// SIMATIC STEP 7 (V5.x) project dry_cooler
// CPU: CPU313(1)
// station: P_ADR_BUS
// station: Hardware
// station: SIMATIC 300 Station
// station: P_ADR_BUS
// station: Configuration
// program: S7 Program(1)

SYMBOL_TABLE
"DBData"	DB 1	DB 1
"DB_Alarm"	DB 2	DB 2	// Db alarmes
"Run Time Animation"	DB 3	DB 3	// Animaçoes
"DBAnalog"	DB 64	DB 64
"DB_Temperature"	DB 100	DB 100	// DB Tratamento analogico
"DB HMI Funtions"	DB 101	DB 101
"Sensores"	FB 105	FB 105
"Analog_Trated"	FC 1	FC 1	// Analog_trated
"Input_Trated"	FC 2	FC 2	// Tratatemto das entradas
"Output_Trated"	FC 3	FC 3	// Tratamento das saidas
"Inputs"	FC 4	FC 4	// Inputs
"Outputs"	FC 5	FC 5	// Outputs
"Pump_Logic"	FC 6	FC 6
"Acionaqamento Ventilador"	FC 7	FC 7
"New Analog"	FC 10	FC 10
"Tratamento_Inputs"	FC 100	FC 100
"Tratamento Saida"	FC 101	FC 101
"SCALE_1"	FC 105	FC 105	// Scaling 1
"Transmissores_Analogicos"	FC 106	FC 106
"SCALE_2"	FC 205	FC 205	// Scaling 2
"Animation_HMI"	FC 255	FC 255
"SCALE_3"	FC 305	FC 305	// Scaling 2
"SCALE_4"	FC 405	FC 405	// Scaling 4
"SCALE_5"	FC 505	FC 505	// Scaling 5
"SCALE_6"	FC 605	FC 605	// Scaling 6
"SCALE_7"	FC 705	FC 705	// Scaling 7
"SCALE_8"	FC 805	FC 805	// Scaling 8
"Pump1_On"	I 4.0	BOOL	// Button On Pump1
"Pump1_Off"	I 4.1	BOOL	// Button Off Pump1
"Pump_2_On"	I 4.2	BOOL	// Button On Pump2
"Puymp2_Off"	I 4.3	BOOL	// Button Off Pump2
"Fan1_On"	I 4.4	BOOL	// Button On Fan1
"Fan1_Off"	I 4.5	BOOL	// Button Off Fan1
"Fan2_On"	I 4.6	BOOL	// Button On Fan2
"Fan2_Off"	I 4.7	BOOL	// Button Off Fan2
"AdiabaticPump_On"	I 5.0	BOOL	// Button On Adb
"AdiabaticPump_Off"	I 5.1	BOOL	// Button Off Adb
"Emergency"	I 5.2	BOOL	// Emergency Button
"Manual"	I 5.3	BOOL	// Manual Switch
"Auto"	I 5.4	BOOL	// Auto Switch
"InSpare1"	I 5.5	BOOL	// Spare 1
"InSpare2"	I 5.6	BOOL	// Spare2
"InSpare3"	I 5.7	BOOL	// Spare3
"CircuitBreakerPump1"	I 8.0	BOOL	// Feedback CB Pump1
"CircuitBrakerPump2"	I 8.1	BOOL	// Feedback CB Pump2
"CircuitBreaker Fan1"	I 8.2	BOOL	// Feedback CB Fan1
"CircuitBraekerFan2"	I 8.3	BOOL	// Feedback CB Fan2
"CircuitBreakerAdbPump"	I 8.4	BOOL	// Feedback CB Adiabatic Pump
"ContactorPump1"	I 8.5	BOOL	// Feedback state contactor pump 1
"ContactorPump2"	I 8.6	BOOL	// Feedback state contactor pump 2
"Contacort.Fan1"	I 8.7	BOOL	// Feedback state contactor fan 1
"ContactorFan2"	I 9.0	BOOL	// Feedback state contactor fan2
"ContactorAdb"	I 9.1	BOOL	// Feedback state contactor adb pump
"FlowSwitch"	I 9.2	BOOL	// Flow Switch signal
"LevelSwitch"	I 9.3	BOOL	// Level switch
"InSpare4"	I 9.4	BOOL	// Spare 4
"InSpare5"	I 9.5	BOOL	// Spare 5
"InSpare6"	I 9.6	BOOL	// Spare 6
"InSpare7"	I 9.7	BOOL	// Spare 7
"Aux_Pump1On"	M 4.0	BOOL	// Aux input pump 1 on
"Aux_Pump1Off"	M 4.1	BOOL	// Aux input pump 1 off
"Aux_Pump2On"	M 4.2	BOOL	// Aux input pump 2 on
"Aux_Pump2Off"	M 4.3	BOOL	// Aux input pump 2 off
"Aux_Fan1On"	M 4.4	BOOL	// Aux input fan 1 on
"Aux_Fan1Off"	M 4.5	BOOL	// Aux input fan 1 off
"Aux_Fan2On"	M 4.6	BOOL	// Aux input fan 2on
"Aux_Fan2Off"	M 4.7	BOOL	// Aux input fan 2 off
"Aux_AdbOn"	M 5.0	BOOL	// Aux input adiabatic on
"Aux_AdbOff"	M 5.1	BOOL	// Aux input adiabatic off
"Aux_Emergency"	M 5.2	BOOL	// Aux input emergency button
"Aux_Manual"	M 5.3	BOOL	// Aux input manual Switch
"Aux_Automatic"	M 5.4	BOOL	// Aux input automatic switch
"Aux_InSpare1"	M 5.5	BOOL	// Aux input spare1
"Aux_InSpare2"	M 5.6	BOOL	// Aux input spare2
"Aux_InSpare3"	M 5.7	BOOL	// Aux input spare3
"Aux_CBPump1"	M 8.0	BOOL	// Aux input circuit breaker pump 1
"Aux_CBPump2"	M 8.1	BOOL	// Aux input circuit breaker pump2
"Aux_CBFan1"	M 8.2	BOOL	// Aux input circuit breaker fan 1
"Aux_CBFan2"	M 8.3	BOOL	// Aux input circuit breaker fan 2
"Aux_CBAdbPump"	M 8.4	BOOL	// Aux input circuit breaker adiabatic
"Aux_FeedPump1"	M 8.5	BOOL	// Aux input feedback contactor pump 1
"Aux_FeedPump2"	M 8.6	BOOL	// Aux input feedback contactor pump 2
"Aux_FeedFan1"	M 8.7	BOOL	// Aux input feedback contactor fan 1
"Aux_FeedFan2"	M 9.0	BOOL	// Aux input feedback contactor fan 2
"Aux_FeedAdbPump"	M 9.1	BOOL	// Aux input feedbcak contactor adiabatic
"Aux_FlowSwitch"	M 9.2	BOOL	// Aux input flow switch
"Aux_LevelSwitch"	M 9.3	BOOL	// Aux input level switch
"Aux_InSpare4"	M 9.4	BOOL	// Aux input spare 4
"Aux_InSpare5"	M 9.5	BOOL	// Aux input spare 5
"Aux_InSpare6"	M 9.6	BOOL	// Aux input spare 6
"Aux_InSpare7"	M 9.7	BOOL	// Auxiliar Input spare 7
"OnAutomaticPump1"	M 10.0	BOOL	// Start pump 1 Automatic
"OnManualPump1"	M 10.1	BOOL	// Start Pump 1 Manual
"Flow Fault"	M 10.2	BOOL	// Water flow in fault pump 1
"Aux_RelayWaterPump1"	M 12.0	BOOL	// Aux out relay pump 1
"Aux_RelayWaterPump2"	M 12.1	BOOL	// Aux out relay pump2
"Aux_RelayFan1"	M 12.2	BOOL	// Aux out relay fan 1
"Aux_RelayFan2"	M 12.3	BOOL	// Aux out relay fan 2
"Aux_RelayAdbPump"	M 12.4	BOOL	// Aux out relay adiabatic pump
"Aux_OutSpare1"	M 12.5	BOOL	// Aux out spare 1
"Aux_OutSpare2"	M 12.6	BOOL	// Aux out spare 2
"Aux_OutSpare3"	M 12.7	BOOL	// Aux out spare 3
"Aux_OutSpare4"	M 13.0	BOOL	// Aux out spare 4
"Aux_OutSpare5"	M 13.1	BOOL	// Aux out spare 5
"Aux_OutSpare6"	M 13.2	BOOL	// Aux out spare 6
"Aux_OutSpare7"	M 13.3	BOOL	// Aux out spare 7
"Aux_HornBuzzer"	M 13.4	BOOL	// Aux out horn buzzer
"Aux_AdiabaticSolenoid"	M 13.5	BOOL	// Aux out adiabatic solenoid
"Aux_LampPump1On"	M 13.6	BOOL	// Aux out lamp pump 1 on
"Aux_LampPump1Fault"	M 13.7	BOOL	// Aux out lamp pump 1 fault
"Aux_LampPump2On"	M 16.0	BOOL	// Aux out lamp pump 2 on
"Aux_LampPump2Fault"	M 16.1	BOOL	// Aux out lamp pump 2 fault
"Aux_LampFan1On"	M 16.2	BOOL	// Aux out lamp fan 1 on
"Aux_LampFan1Fault"	M 16.3	BOOL	// Aux out lamp fan 1 fault
"Aux_LampFan2On"	M 16.4	BOOL	// Aux out lamp fan 2 on
"Aux_LampFan2Fault"	M 16.5	BOOL	// Aux out lamp fan 2 fault
"Aux_LampAdiabaticOn"	M 16.6	BOOL	// Aux out lamp adiabatic on
"Aux_LampAdiabaticFault"	M 16.7	BOOL	// Aux out lamp adiabatic fault
"DI_Input"	MW 2	WORD
"R_Input"	MW 4	WORD
"Cycle Execution"	OB 1	OB 1
"Loss of Rack Fault"	OB 86	OB 86
"Complete Restart"	OB 100	OB 100
"Temp_Input"	PIW 256	WORD	// Temp_Input
"Temp_Output"	PIW 258	WORD	// Temp_Output
"RelayWaterPump1"	Q 12.0	BOOL	// Relay water pum 1
"RelayWaterPump2"	Q 12.1	BOOL	// Relay water Pump 2
"RelayFan1"	Q 12.2	BOOL	// Relay fan 1
"RelayFan2"	Q 12.3	BOOL	// Relay fan 2
"RelayAdiabaticPump"	Q 12.4	BOOL	// Relay adiabatic pump
"OutSpare1"	Q 12.5	BOOL	// Out Spare1
"OutSpare2"	Q 12.6	BOOL	// Out Spare 2
"OutSpare3"	Q 12.7	BOOL	// Out Spare 3
"OutSpare4"	Q 13.0	BOOL	// Out Spare 4
"OutSpare5"	Q 13.1	BOOL	// Out Spare 5
"OutSpare6"	Q 13.2	BOOL	// Out Spare 6
"OutSpare7"	Q 13.3	BOOL	// Out Spare 7
"HornBuzzer"	Q 13.4	BOOL	// Horn Buzzer
"RelayAdbSolenoid"	Q 13.5	BOOL	// Relay adiabatic solenoid
"LightOnPump1"	Q 13.6	BOOL	// Light on pump 1
"LightFaultPump1"	Q 13.7	BOOL	// Light fault pump 1
"LightOnPump2"	Q 16.0	BOOL	// Light on pump 2
"LightFaultPump2"	Q 16.1	BOOL	// Light fault pump 2
"LightOnFan1"	Q 16.2	BOOL	// Light on fan 1
"LightFaultFan1"	Q 16.3	BOOL	// Light fault fan 1
"LightOnFan2"	Q 16.4	BOOL	// Light on fan 2
"LightFaultFan2"	Q 16.5	BOOL	// Light fault fan 2
"LightOnAdb"	Q 16.6	BOOL	// Light on adiabatic
"LightFaultAdb"	Q 16.7	BOOL	// Light fault adiabatic
"Timer Water Flow"	T 0	TIMER
"Factor And ValueSensor"	VAT 1	
END_SYMBOL_TABLE

FUNCTION "Analog_Trated" : VOID	// FC 1
VERSION : 0.1
BEGIN
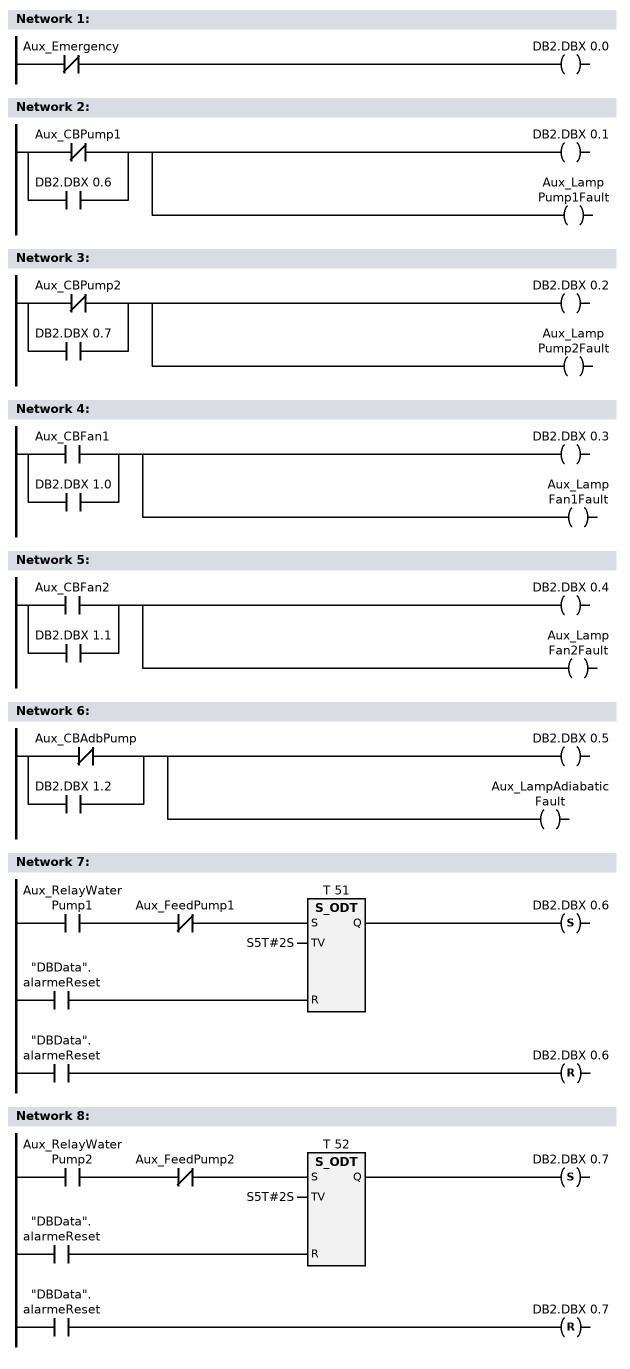
NETWORK
TITLE =
      AN    "Aux_Emergency";
      =     DB2.DBX 0.0;
NETWORK
TITLE =
      ON    "Aux_CBPump1";
      O     DB2.DBX 0.6;
      =     DB2.DBX 0.1;
      =     "Aux_LampPump1Fault";
NETWORK
TITLE =
      ON    "Aux_CBPump2";
      O     DB2.DBX 0.7;
      =     DB2.DBX 0.2;
      =     "Aux_LampPump2Fault";
NETWORK
TITLE =
      O     "Aux_CBFan1";
      O     DB2.DBX 1.0;
      =     DB2.DBX 0.3;
      =     "Aux_LampFan1Fault";
NETWORK
TITLE =
      O     "Aux_CBFan2";
      O     DB2.DBX 1.1;
      =     DB2.DBX 0.4;
      =     "Aux_LampFan2Fault";
NETWORK
TITLE =
      ON    "Aux_CBAdbPump";
      O     DB2.DBX 1.2;
      =     DB2.DBX 0.5;
      =     "Aux_LampAdiabaticFault";
NETWORK
TITLE =
      A(;
      A     "Aux_RelayWaterPump1";
      AN    "Aux_FeedPump1";
      L     S5T#2S;
      SD    T 51;
      A     "DBData".alarmeReset;
      R     T 51;
      NOP   0;
      NOP   0;
      A     T 51;
      );
      S     DB2.DBX 0.6;
      A     "DBData".alarmeReset;
      R     DB2.DBX 0.6;
      NOP   0;
NETWORK
TITLE =
      A(;
      A     "Aux_RelayWaterPump2";
      AN    "Aux_FeedPump2";
      L     S5T#2S;
      SD    T 52;
      A     "DBData".alarmeReset;
      R     T 52;
      NOP   0;
      NOP   0;
      A     T 52;
      );
      S     DB2.DBX 0.7;
      A     "DBData".alarmeReset;
      R     DB2.DBX 0.7;
      NOP   0;
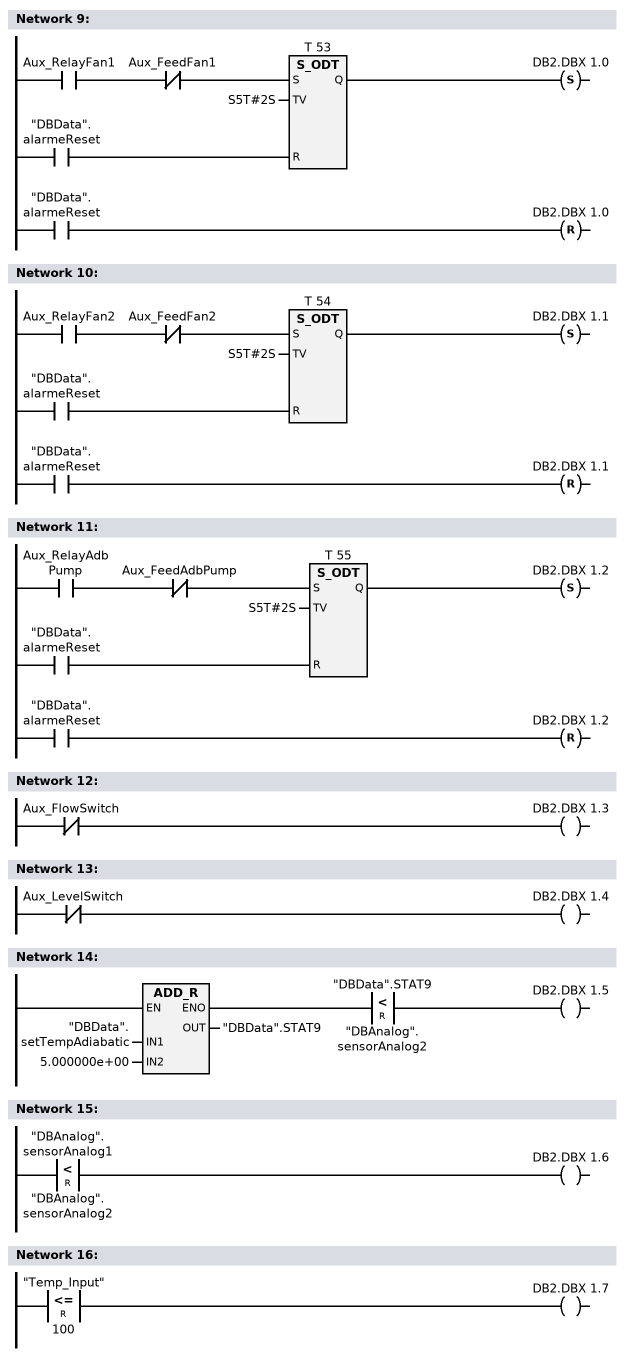
NETWORK
TITLE =
      A(;
      A     "Aux_RelayFan1";
      AN    "Aux_FeedFan1";
      L     S5T#2S;
      SD    T 53;
      A     "DBData".alarmeReset;
      R     T 53;
      NOP   0;
      NOP   0;
      A     T 53;
      );
      S     DB2.DBX 1.0;
      A     "DBData".alarmeReset;
      R     DB2.DBX 1.0;
      NOP   0;
NETWORK
TITLE =
      A(;
      A     "Aux_RelayFan2";
      AN    "Aux_FeedFan2";
      L     S5T#2S;
      SD    T 54;
      A     "DBData".alarmeReset;
      R     T 54;
      NOP   0;
      NOP   0;
      A     T 54;
      );
      S     DB2.DBX 1.1;
      A     "DBData".alarmeReset;
      R     DB2.DBX 1.1;
      NOP   0;
NETWORK
TITLE =
      A(;
      A     "Aux_RelayAdbPump";
      AN    "Aux_FeedAdbPump";
      L     S5T#2S;
      SD    T 55;
      A     "DBData".alarmeReset;
      R     T 55;
      NOP   0;
      NOP   0;
      A     T 55;
      );
      S     DB2.DBX 1.2;
      A     "DBData".alarmeReset;
      R     DB2.DBX 1.2;
      NOP   0;
NETWORK
TITLE =
      AN    "Aux_FlowSwitch";
      =     DB2.DBX 1.3;
NETWORK
TITLE =
      AN    "Aux_LevelSwitch";
      =     DB2.DBX 1.4;
NETWORK
TITLE =
      A(;
      L     "DBData".setTempAdiabatic;
      L     5.000000e+00;
      +R;
      T     "DBData".STAT9;
      AN    OV;
      SAVE;
      CLR;
      A     BR;
      );
      A(;
      L     "DBData".STAT9;
      L     "DBAnalog".sensorAnalog2;
      <R;
      );
      =     DB2.DBX 1.5;
NETWORK
TITLE =
      L     "DBAnalog".sensorAnalog1;
      L     "DBAnalog".sensorAnalog2;
      <R;
      =     DB2.DBX 1.6;
NETWORK
TITLE =
      L     "Temp_Input";
      L     100;
      <=R;
      =     DB2.DBX 1.7;
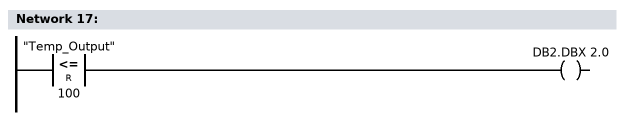
NETWORK
TITLE =
      L     "Temp_Output";
      L     100;
      <=R;
      =     DB2.DBX 2.0;
END_FUNCTION

FUNCTION "Input_Trated" : VOID	// FC 2
NAME : Inputs
VERSION : 0.1
BEGIN
// (block stored without names or comments; labels and parameter names are numbered)
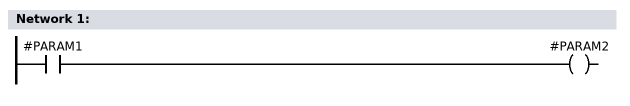
NETWORK
TITLE =
      A     #PARAM1;
      =     #PARAM2;
END_FUNCTION

FUNCTION "Output_Trated" : VOID	// FC 3
VERSION : 0.1
BEGIN
// (block stored without names or comments; labels and parameter names are numbered)
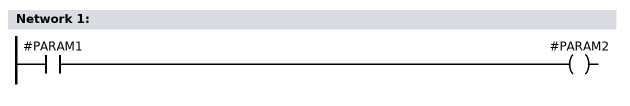
NETWORK
TITLE =
      A     #PARAM1;
      =     #PARAM2;
END_FUNCTION

FUNCTION "Inputs" : VOID	// FC 4
VERSION : 0.1
BEGIN
// (block stored without names or comments; labels and parameter names are numbered)
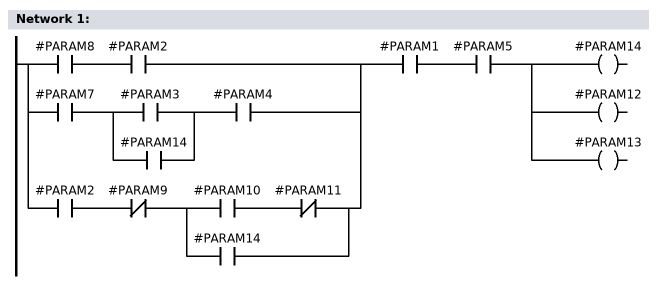
NETWORK
TITLE =
      A(;
      A     #PARAM8;
      A     #PARAM2;
      O;
      A     #PARAM7;
      A(;
      O     #PARAM3;
      O     #PARAM14;
      );
      A     #PARAM4;
      O;
      A     #PARAM2;
      AN    #PARAM9;
      A(;
      A     #PARAM10;
      AN    #PARAM11;
      O     #PARAM14;
      );
      );
      A     #PARAM1;
      A     #PARAM5;
      =     #PARAM14;
      =     #PARAM12;
      =     #PARAM13;
END_FUNCTION

FUNCTION "Outputs" : VOID	// FC 5
VERSION : 0.1
BEGIN
// (block stored without names or comments; labels and parameter names are numbered)
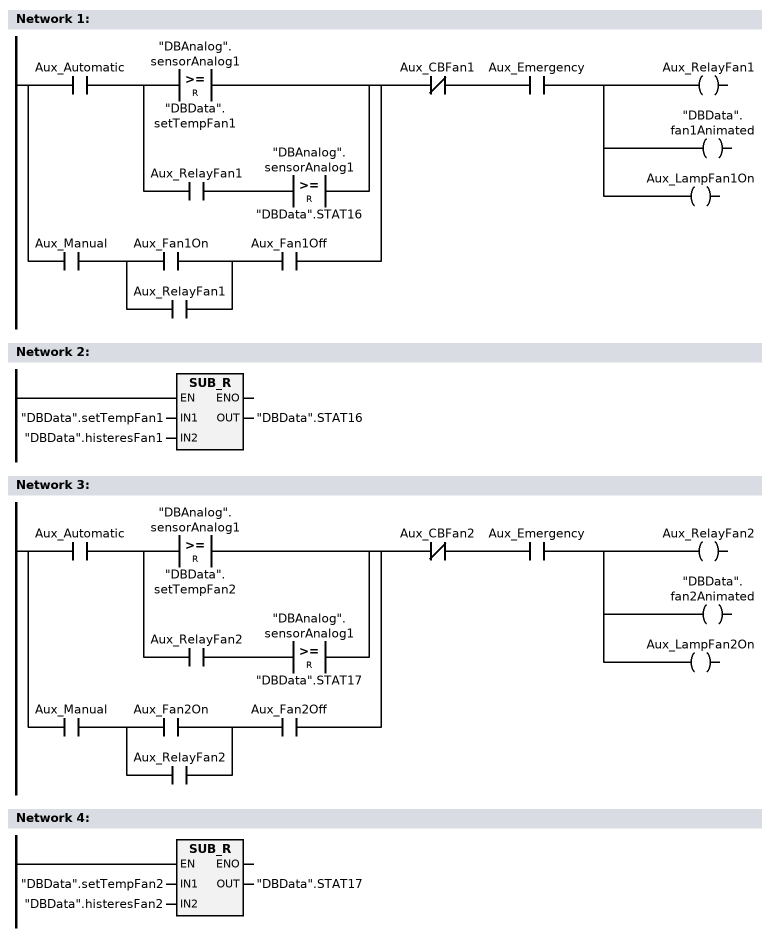
NETWORK
TITLE =
      A(;
      A     "Aux_Automatic";
      A(;
      O(;
      L     "DBAnalog".sensorAnalog1;
      L     "DBData".setTempFan1;
      >=R;
      );
      O;
      A     "Aux_RelayFan1";
      A(;
      L     "DBAnalog".sensorAnalog1;
      L     "DBData".STAT16;
      >=R;
      );
      );
      O;
      A     "Aux_Manual";
      A(;
      O     "Aux_Fan1On";
      O     "Aux_RelayFan1";
      );
      A     "Aux_Fan1Off";
      );
      AN    "Aux_CBFan1";
      A     "Aux_Emergency";
      =     "Aux_RelayFan1";
      =     "DBData".fan1Animated;
      =     "Aux_LampFan1On";
NETWORK
TITLE =
      L     "DBData".setTempFan1;
      L     "DBData".histeresFan1;
      -R;
      T     "DBData".STAT16;
      NOP   0;
NETWORK
TITLE =
      A(;
      A     "Aux_Automatic";
      A(;
      O(;
      L     "DBAnalog".sensorAnalog1;
      L     "DBData".setTempFan2;
      >=R;
      );
      O;
      A     "Aux_RelayFan2";
      A(;
      L     "DBAnalog".sensorAnalog1;
      L     "DBData".STAT17;
      >=R;
      );
      );
      O;
      A     "Aux_Manual";
      A(;
      O     "Aux_Fan2On";
      O     "Aux_RelayFan2";
      );
      A     "Aux_Fan2Off";
      );
      AN    "Aux_CBFan2";
      A     "Aux_Emergency";
      =     "Aux_RelayFan2";
      =     "DBData".fan2Animated;
      =     "Aux_LampFan2On";
NETWORK
TITLE =
      L     "DBData".setTempFan2;
      L     "DBData".histeresFan2;
      -R;
      T     "DBData".STAT17;
      NOP   0;
END_FUNCTION

FUNCTION "Pump_Logic" : VOID	// FC 6
VERSION : 0.1
BEGIN
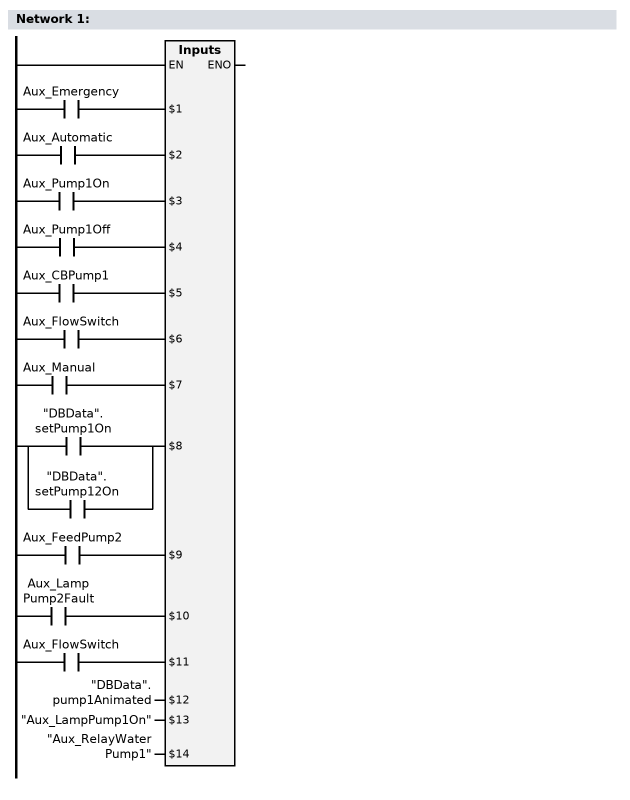
NETWORK
TITLE =
      A     "Aux_Emergency";
      =     L 0.0;
      BLD   103;
      A     "Aux_Automatic";
      =     L 0.1;
      BLD   103;
      A     "Aux_Pump1On";
      =     L 0.2;
      BLD   103;
      A     "Aux_Pump1Off";
      =     L 0.3;
      BLD   103;
      A     "Aux_CBPump1";
      =     L 0.4;
      BLD   103;
      A     "Aux_FlowSwitch";
      =     L 0.5;
      BLD   103;
      A     "Aux_Manual";
      =     L 0.6;
      BLD   103;
      A(;
      O     "DBData".setPump1On;
      O     "DBData".setPump12On;
      );
      =     L 0.7;
      BLD   103;
      A     "Aux_FeedPump2";
      =     L 1.0;
      BLD   103;
      A     "Aux_LampPump2Fault";
      =     L 1.1;
      BLD   103;
      A     "Aux_FlowSwitch";
      =     L 1.2;
      BLD   103;
      CALL  "Inputs" (
           $1                       := L 0.0,
           $2                       := L 0.1,
           $3                       := L 0.2,
           $4                       := L 0.3,
           $5                       := L 0.4,
           $6                       := L 0.5,
           $7                       := L 0.6,
           $8                       := L 0.7,
           $9                       := L 1.0,
           $10                      := L 1.1,
           $11                      := L 1.2,
           $12                      := "DBData".pump1Animated,
           $13                      := "Aux_LampPump1On",
           $14                      := "Aux_RelayWaterPump1");
      NOP   0;
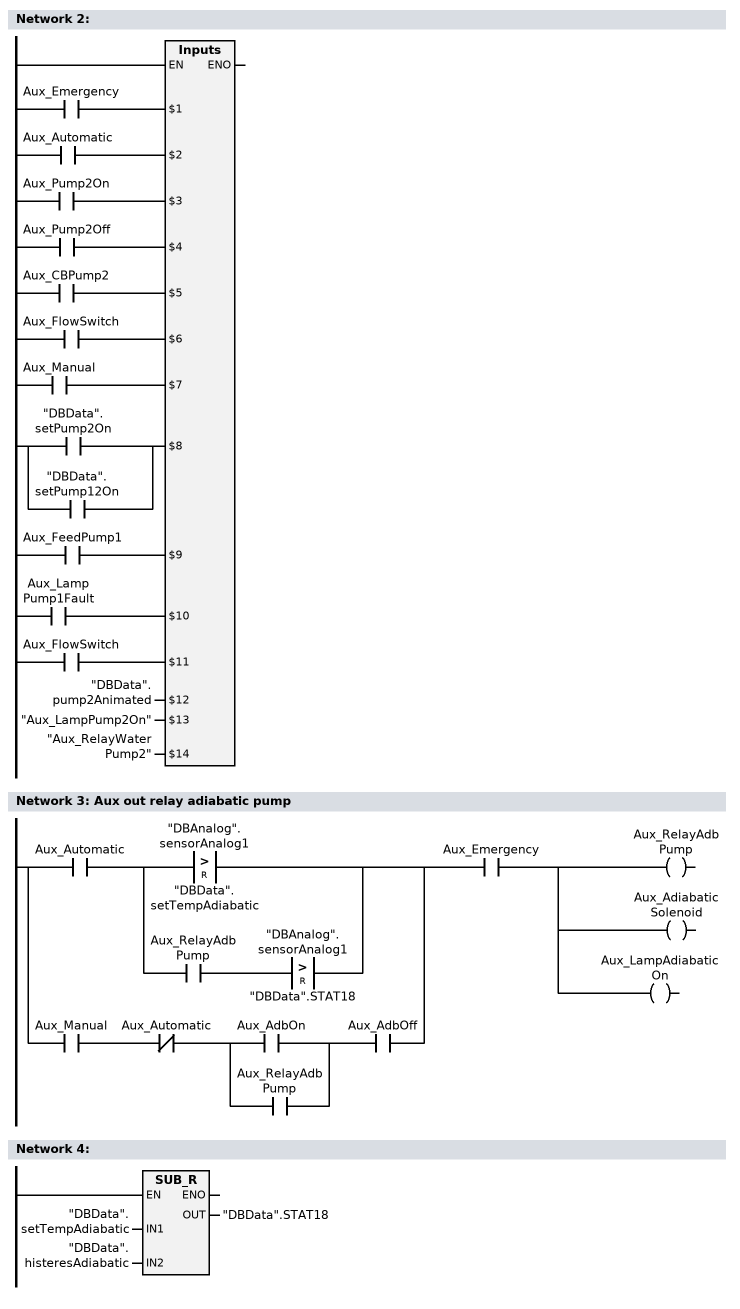
NETWORK
TITLE =
      A     "Aux_Emergency";
      =     L 0.0;
      BLD   103;
      A     "Aux_Automatic";
      =     L 0.1;
      BLD   103;
      A     "Aux_Pump2On";
      =     L 0.2;
      BLD   103;
      A     "Aux_Pump2Off";
      =     L 0.3;
      BLD   103;
      A     "Aux_CBPump2";
      =     L 0.4;
      BLD   103;
      A     "Aux_FlowSwitch";
      =     L 0.5;
      BLD   103;
      A     "Aux_Manual";
      =     L 0.6;
      BLD   103;
      A(;
      O     "DBData".setPump2On;
      O     "DBData".setPump12On;
      );
      =     L 0.7;
      BLD   103;
      A     "Aux_FeedPump1";
      =     L 1.0;
      BLD   103;
      A     "Aux_LampPump1Fault";
      =     L 1.1;
      BLD   103;
      A     "Aux_FlowSwitch";
      =     L 1.2;
      BLD   103;
      CALL  "Inputs" (
           $1                       := L 0.0,
           $2                       := L 0.1,
           $3                       := L 0.2,
           $4                       := L 0.3,
           $5                       := L 0.4,
           $6                       := L 0.5,
           $7                       := L 0.6,
           $8                       := L 0.7,
           $9                       := L 1.0,
           $10                      := L 1.1,
           $11                      := L 1.2,
           $12                      := "DBData".pump2Animated,
           $13                      := "Aux_LampPump2On",
           $14                      := "Aux_RelayWaterPump2");
      NOP   0;
NETWORK
TITLE = Aux out relay adiabatic pump
      A(;
      A     "Aux_Automatic";
      A(;
      O(;
      L     "DBAnalog".sensorAnalog1;
      L     "DBData".setTempAdiabatic;
      >R;
      );
      O;
      A     "Aux_RelayAdbPump";
      A(;
      L     "DBAnalog".sensorAnalog1;
      L     "DBData".STAT18;
      >R;
      );
      );
      O;
      A     "Aux_Manual";
      AN    "Aux_Automatic";
      A(;
      O     "Aux_AdbOn";
      O     "Aux_RelayAdbPump";
      );
      A     "Aux_AdbOff";
      );
      A     "Aux_Emergency";
      =     "Aux_RelayAdbPump";
      =     "Aux_AdiabaticSolenoid";
      =     "Aux_LampAdiabaticOn";
NETWORK
TITLE =
      L     "DBData".setTempAdiabatic;
      L     "DBData".histeresAdiabatic;
      -R;
      T     "DBData".STAT18;
      NOP   0;
END_FUNCTION

FUNCTION "Acionaqamento Ventilador" : VOID	// FC 7
VERSION : 0.1
BEGIN
// (block stored without names or comments; labels and parameter names are numbered)
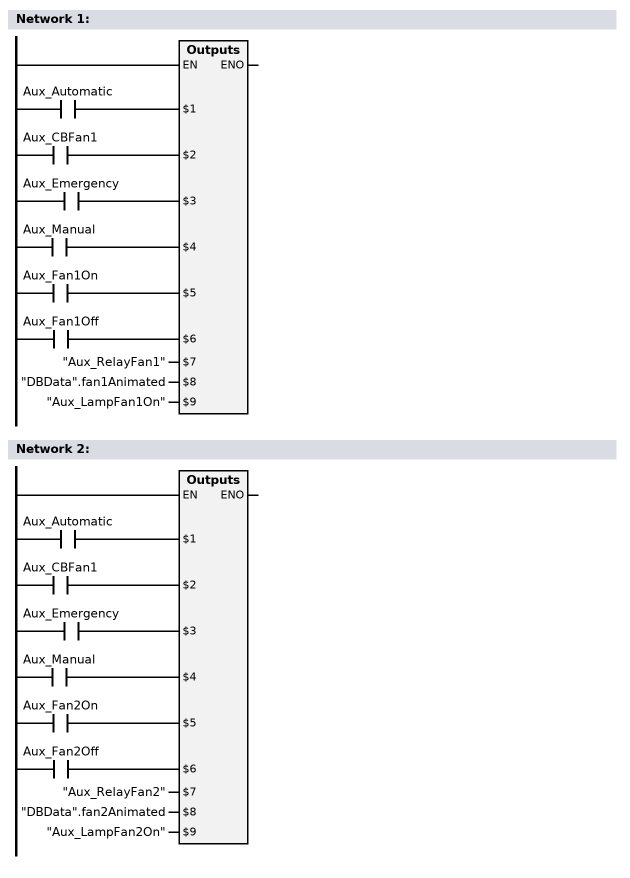
NETWORK
TITLE =
      A     "Aux_Automatic";
      =     L 0.0;
      BLD   103;
      A     "Aux_CBFan1";
      =     L 0.1;
      BLD   103;
      A     "Aux_Emergency";
      =     L 0.2;
      BLD   103;
      A     "Aux_Manual";
      =     L 0.3;
      BLD   103;
      A     "Aux_Fan1On";
      =     L 0.4;
      BLD   103;
      A     "Aux_Fan1Off";
      =     L 0.5;
      BLD   103;
      CALL  "Outputs" (
           $1                       := L 0.0,
           $2                       := L 0.1,
           $3                       := L 0.2,
           $4                       := L 0.3,
           $5                       := L 0.4,
           $6                       := L 0.5,
           $7                       := "Aux_RelayFan1",
           $8                       := "DBData".fan1Animated,
           $9                       := "Aux_LampFan1On");
      NOP   0;
NETWORK
TITLE =
      A     "Aux_Automatic";
      =     L 0.0;
      BLD   103;
      A     "Aux_CBFan1";
      =     L 0.1;
      BLD   103;
      A     "Aux_Emergency";
      =     L 0.2;
      BLD   103;
      A     "Aux_Manual";
      =     L 0.3;
      BLD   103;
      A     "Aux_Fan2On";
      =     L 0.4;
      BLD   103;
      A     "Aux_Fan2Off";
      =     L 0.5;
      BLD   103;
      CALL  "Outputs" (
           $1                       := L 0.0,
           $2                       := L 0.1,
           $3                       := L 0.2,
           $4                       := L 0.3,
           $5                       := L 0.4,
           $6                       := L 0.5,
           $7                       := "Aux_RelayFan2",
           $8                       := "DBData".fan2Animated,
           $9                       := "Aux_LampFan2On");
      NOP   0;
END_FUNCTION

FUNCTION FC 8 : VOID
VERSION : 0.1
BEGIN
// (block stored without names or comments; labels and parameter names are numbered)
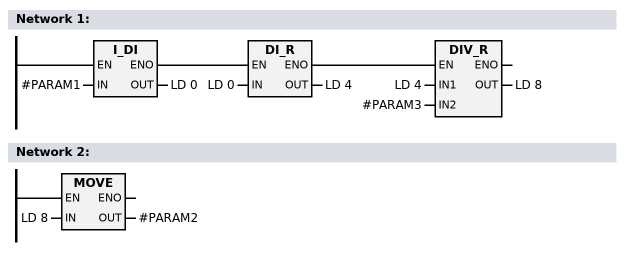
NETWORK
TITLE =
      A(;
      A(;
      L     #PARAM1;
      ITD;
      T     LD 0;
      SET;
      SAVE;
      CLR;
      A     BR;
      );
      JNB   M001;
      L     LD 0;
      DTR;
      T     LD 4;
      SET;
      SAVE;
      CLR;
M001: A     BR;
      );
      JNB   M002;
      L     LD 4;
      L     #PARAM3;
      /R;
      T     LD 8;
M002: NOP   0;
NETWORK
TITLE =
      L     LD 8;
      T     #PARAM2;
      NOP   0;
END_FUNCTION

FUNCTION FC 9 : VOID
VERSION : 0.1
BEGIN
// (block stored without names or comments; labels and parameter names are numbered)
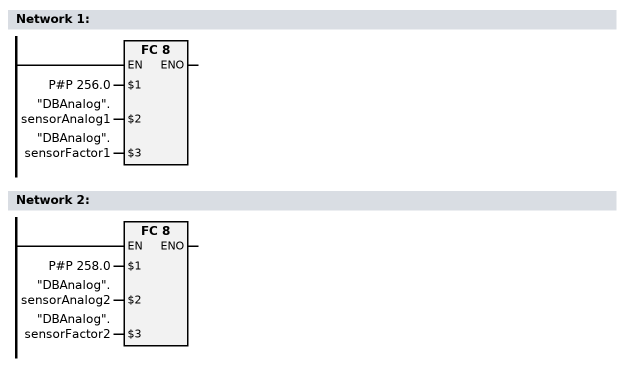
NETWORK
TITLE =
      CALL  FC 8 (
           $1                       := P#P 256.0,
           $2                       := "DBAnalog".sensorAnalog1,
           $3                       := "DBAnalog".sensorFactor1);
      NOP   0;
NETWORK
TITLE =
      CALL  FC 8 (
           $1                       := P#P 258.0,
           $2                       := "DBAnalog".sensorAnalog2,
           $3                       := "DBAnalog".sensorFactor2);
      NOP   0;
END_FUNCTION

FUNCTION "New Analog" : VOID	// FC 10
VERSION : 0.1
BEGIN
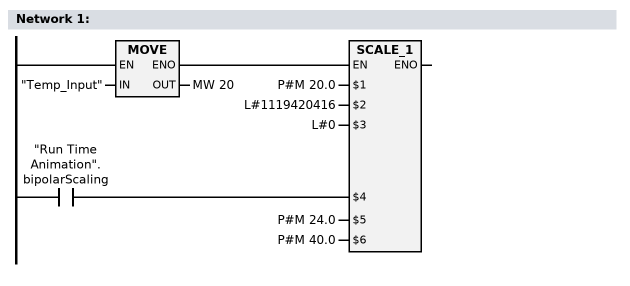
NETWORK
TITLE =
      A     "Run Time Animation".bipolarScaling;
      =     L 0.0;
      BLD   103;
      A(;
      L     "Temp_Input";
      T     MW 20;
      SET;
      SAVE;
      CLR;
      A     BR;
      );
      JNB   _001;
      CALL  "SCALE_1" (
           $1                       := P#M 20.0,
           $2                       := L#1119420416,
           $3                       := L#0,
           $4                       := L 0.0,
           $5                       := P#M 24.0,
           $6                       := P#M 40.0);
_001: NOP   0;
NETWORK
TITLE =
END_FUNCTION

FUNCTION FC 95 : VOID
VERSION : 0.1
BEGIN
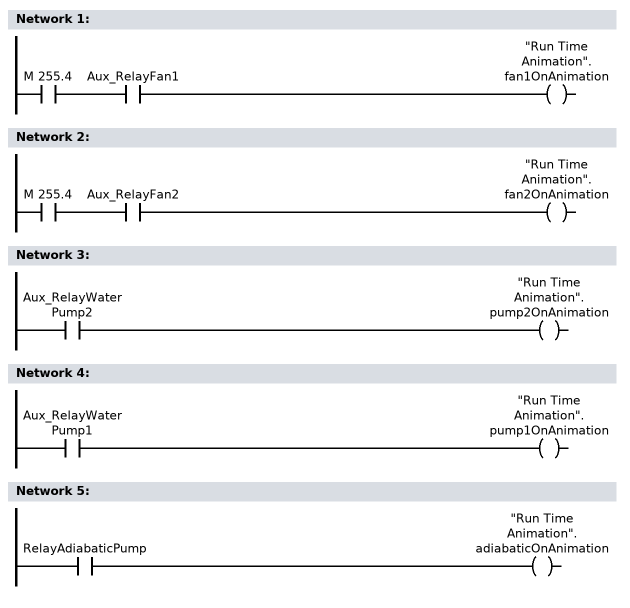
NETWORK
TITLE =
      A     M 255.4;
      A     "Aux_RelayFan1";
      =     "Run Time Animation".fan1OnAnimation;
NETWORK
TITLE =
      A     M 255.4;
      A     "Aux_RelayFan2";
      =     "Run Time Animation".fan2OnAnimation;
NETWORK
TITLE =
      A     "Aux_RelayWaterPump2";
      =     "Run Time Animation".pump2OnAnimation;
NETWORK
TITLE =
      A     "Aux_RelayWaterPump1";
      =     "Run Time Animation".pump1OnAnimation;
NETWORK
TITLE =
      A     "RelayAdiabaticPump";
      =     "Run Time Animation".adiabaticOnAnimation;
END_FUNCTION

FUNCTION "Tratamento_Inputs" : VOID	// FC 100
VERSION : 0.1
BEGIN
// (block stored without names or comments; labels and parameter names are numbered)
NETWORK
TITLE =
      A     "Pump1_On";
      =     L 0.0;
      BLD   103;
      CALL  "Input_Trated" (
           $1                       := L 0.0,
           $2                       := P#M 4.0);
      NOP   0;
NETWORK
TITLE =
      A     "Pump1_Off";
      =     L 0.0;
      BLD   103;
      CALL  "Input_Trated" (
           $1                       := L 0.0,
           $2                       := "Aux_Pump1Off");
      NOP   0;
NETWORK
TITLE =
      A     "Pump_2_On";
      =     L 0.0;
      BLD   103;
      CALL  "Input_Trated" (
           $1                       := L 0.0,
           $2                       := "Aux_Pump2On");
      NOP   0;
NETWORK
TITLE =
      A     "Puymp2_Off";
      =     L 0.0;
      BLD   103;
      CALL  "Input_Trated" (
           $1                       := L 0.0,
           $2                       := "Aux_Pump2Off");
      NOP   0;
NETWORK
TITLE =
      A     "Fan1_On";
      =     L 0.0;
      BLD   103;
      CALL  "Input_Trated" (
           $1                       := L 0.0,
           $2                       := "Aux_Fan1On");
      NOP   0;
NETWORK
TITLE =
      A     "Fan1_Off";
      =     L 0.0;
      BLD   103;
      CALL  "Input_Trated" (
           $1                       := L 0.0,
           $2                       := "Aux_Fan1Off");
      NOP   0;
NETWORK
TITLE =
      A     "Fan2_On";
      =     L 0.0;
      BLD   103;
      CALL  "Input_Trated" (
           $1                       := L 0.0,
           $2                       := "Aux_Fan2On");
      NOP   0;
NETWORK
TITLE =
      A     "Fan2_Off";
      =     L 0.0;
      BLD   103;
      CALL  "Input_Trated" (
           $1                       := L 0.0,
           $2                       := "Aux_Fan2Off");
      NOP   0;
NETWORK
TITLE =
      A     "AdiabaticPump_On";
      =     L 0.0;
      BLD   103;
      CALL  "Input_Trated" (
           $1                       := L 0.0,
           $2                       := "Aux_AdbOn");
      NOP   0;
NETWORK
TITLE =
      A     "AdiabaticPump_Off";
      =     L 0.0;
      BLD   103;
      CALL  "Input_Trated" (
           $1                       := L 0.0,
           $2                       := "Aux_AdbOff");
      NOP   0;
NETWORK
TITLE =
      A     "Emergency";
      =     L 0.0;
      BLD   103;
      CALL  "Input_Trated" (
           $1                       := L 0.0,
           $2                       := "Aux_Emergency");
      NOP   0;
NETWORK
TITLE =
      A     "Manual";
      =     L 0.0;
      BLD   103;
      CALL  "Input_Trated" (
           $1                       := L 0.0,
           $2                       := "Aux_Manual");
      NOP   0;
NETWORK
TITLE =
      A     "Auto";
      =     L 0.0;
      BLD   103;
      CALL  "Input_Trated" (
           $1                       := L 0.0,
           $2                       := "Aux_Automatic");
      NOP   0;
NETWORK
TITLE =
      A     "InSpare1";
      =     L 0.0;
      BLD   103;
      CALL  "Input_Trated" (
           $1                       := L 0.0,
           $2                       := "Aux_InSpare1");
      NOP   0;
NETWORK
TITLE =
      A     "InSpare2";
      =     L 0.0;
      BLD   103;
      CALL  "Input_Trated" (
           $1                       := L 0.0,
           $2                       := "Aux_InSpare2");
      NOP   0;
NETWORK
TITLE =
      A     "InSpare3";
      =     L 0.0;
      BLD   103;
      CALL  "Input_Trated" (
           $1                       := L 0.0,
           $2                       := "Aux_InSpare3");
      NOP   0;
NETWORK
TITLE =
      A     "CircuitBreakerPump1";
      =     L 0.0;
      BLD   103;
      CALL  "Input_Trated" (
           $1                       := L 0.0,
           $2                       := "Aux_CBPump1");
      NOP   0;
NETWORK
TITLE =
      A     "CircuitBrakerPump2";
      =     L 0.0;
      BLD   103;
      CALL  "Input_Trated" (
           $1                       := L 0.0,
           $2                       := "Aux_CBPump2");
      NOP   0;
NETWORK
TITLE =
      A     "CircuitBreaker Fan1";
      =     L 0.0;
      BLD   103;
      CALL  "Input_Trated" (
           $1                       := L 0.0,
           $2                       := "Aux_CBFan1");
      NOP   0;
NETWORK
TITLE =
      A     "CircuitBraekerFan2";
      =     L 0.0;
      BLD   103;
      CALL  "Input_Trated" (
           $1                       := L 0.0,
           $2                       := "Aux_CBFan2");
      NOP   0;
NETWORK
TITLE =
      A     "CircuitBreakerAdbPump";
      =     L 0.0;
      BLD   103;
      CALL  "Input_Trated" (
           $1                       := L 0.0,
           $2                       := "Aux_CBAdbPump");
      NOP   0;
NETWORK
TITLE =
      A     "ContactorPump1";
      =     L 0.0;
      BLD   103;
      CALL  "Input_Trated" (
           $1                       := L 0.0,
           $2                       := "Aux_FeedPump1");
      NOP   0;
NETWORK
TITLE =
      A     "ContactorPump2";
      =     L 0.0;
      BLD   103;
      CALL  "Input_Trated" (
           $1                       := L 0.0,
           $2                       := "Aux_FeedPump2");
      NOP   0;
NETWORK
TITLE =
      A     "Contacort.Fan1";
      =     L 0.0;
      BLD   103;
      CALL  "Input_Trated" (
           $1                       := L 0.0,
           $2                       := "Aux_FeedFan1");
      NOP   0;
NETWORK
TITLE =
      A     "ContactorFan2";
      =     L 0.0;
      BLD   103;
      CALL  "Input_Trated" (
           $1                       := L 0.0,
           $2                       := "Aux_FeedFan2");
      NOP   0;
NETWORK
TITLE =
      A     "ContactorAdb";
      =     L 0.0;
      BLD   103;
      CALL  "Input_Trated" (
           $1                       := L 0.0,
           $2                       := "Aux_FeedAdbPump");
      NOP   0;
NETWORK
TITLE =
      A     "FlowSwitch";
      =     L 0.0;
      BLD   103;
      CALL  "Input_Trated" (
           $1                       := L 0.0,
           $2                       := "Aux_FlowSwitch");
      NOP   0;
NETWORK
TITLE =
      A     "LevelSwitch";
      =     L 0.0;
      BLD   103;
      CALL  "Input_Trated" (
           $1                       := L 0.0,
           $2                       := "Aux_LevelSwitch");
      NOP   0;
NETWORK
TITLE =
      A     "InSpare4";
      =     L 0.0;
      BLD   103;
      CALL  "Input_Trated" (
           $1                       := L 0.0,
           $2                       := "Aux_InSpare4");
      NOP   0;
NETWORK
TITLE =
      A     "InSpare5";
      =     L 0.0;
      BLD   103;
      CALL  "Input_Trated" (
           $1                       := L 0.0,
           $2                       := "Aux_InSpare5");
      NOP   0;
NETWORK
TITLE =
      A     "InSpare6";
      =     L 0.0;
      BLD   103;
      CALL  "Input_Trated" (
           $1                       := L 0.0,
           $2                       := "Aux_InSpare6");
      NOP   0;
NETWORK
TITLE =
      A     "InSpare7";
      =     L 0.0;
      BLD   103;
      CALL  "Input_Trated" (
           $1                       := L 0.0,
           $2                       := "Aux_InSpare7");
      NOP   0;
END_FUNCTION

FUNCTION "Tratamento Saida" : VOID	// FC 101
VERSION : 0.1
BEGIN
// (block stored without names or comments; labels and parameter names are numbered)
NETWORK
TITLE =
      A     "Aux_RelayWaterPump1";
      =     L 0.0;
      BLD   103;
      CALL  "Output_Trated" (
           $1                       := L 0.0,
           $2                       := "RelayWaterPump1");
      NOP   0;
NETWORK
TITLE =
      A     "Aux_RelayWaterPump2";
      =     L 0.0;
      BLD   103;
      CALL  "Output_Trated" (
           $1                       := L 0.0,
           $2                       := "RelayWaterPump2");
      NOP   0;
NETWORK
TITLE =
      A     "Aux_RelayFan1";
      =     L 0.0;
      BLD   103;
      CALL  "Output_Trated" (
           $1                       := L 0.0,
           $2                       := "RelayFan1");
      NOP   0;
NETWORK
TITLE =
      A     "Aux_RelayFan2";
      =     L 0.0;
      BLD   103;
      CALL  "Output_Trated" (
           $1                       := L 0.0,
           $2                       := "RelayFan2");
      NOP   0;
NETWORK
TITLE =
      A     "Aux_RelayAdbPump";
      =     L 0.0;
      BLD   103;
      CALL  "Output_Trated" (
           $1                       := L 0.0,
           $2                       := "RelayAdiabaticPump");
      NOP   0;
NETWORK
TITLE =
      A     "Aux_OutSpare1";
      =     L 0.0;
      BLD   103;
      CALL  "Output_Trated" (
           $1                       := L 0.0,
           $2                       := "OutSpare1");
      NOP   0;
NETWORK
TITLE =
      A     "Aux_OutSpare2";
      =     L 0.0;
      BLD   103;
      CALL  "Output_Trated" (
           $1                       := L 0.0,
           $2                       := "OutSpare2");
      NOP   0;
NETWORK
TITLE =
      A     "Aux_OutSpare3";
      =     L 0.0;
      BLD   103;
      CALL  "Output_Trated" (
           $1                       := L 0.0,
           $2                       := "OutSpare3");
      NOP   0;
NETWORK
TITLE =
      A     "Aux_OutSpare4";
      =     L 0.0;
      BLD   103;
      CALL  "Output_Trated" (
           $1                       := L 0.0,
           $2                       := "OutSpare4");
      NOP   0;
NETWORK
TITLE =
      A     "Aux_OutSpare5";
      =     L 0.0;
      BLD   103;
      CALL  "Output_Trated" (
           $1                       := L 0.0,
           $2                       := "OutSpare5");
      NOP   0;
NETWORK
TITLE =
      A     "Aux_OutSpare6";
      =     L 0.0;
      BLD   103;
      CALL  "Output_Trated" (
           $1                       := L 0.0,
           $2                       := "OutSpare6");
      NOP   0;
NETWORK
TITLE =
      A     "Aux_OutSpare7";
      =     L 0.0;
      BLD   103;
      CALL  "Output_Trated" (
           $1                       := L 0.0,
           $2                       := "OutSpare7");
      NOP   0;
NETWORK
TITLE =
      A     "Aux_HornBuzzer";
      =     L 0.0;
      BLD   103;
      CALL  "Output_Trated" (
           $1                       := L 0.0,
           $2                       := "HornBuzzer");
      NOP   0;
NETWORK
TITLE =
      A     "Aux_AdiabaticSolenoid";
      =     L 0.0;
      BLD   103;
      CALL  "Output_Trated" (
           $1                       := L 0.0,
           $2                       := "RelayAdbSolenoid");
      NOP   0;
NETWORK
TITLE =
      A     "Aux_LampPump1On";
      =     L 0.0;
      BLD   103;
      CALL  "Output_Trated" (
           $1                       := L 0.0,
           $2                       := "LightOnPump1");
      NOP   0;
NETWORK
TITLE =
      A     "Aux_LampPump1Fault";
      =     L 0.0;
      BLD   103;
      CALL  "Output_Trated" (
           $1                       := L 0.0,
           $2                       := "LightFaultPump1");
      NOP   0;
NETWORK
TITLE =
      A     "Aux_LampPump2On";
      =     L 0.0;
      BLD   103;
      CALL  "Output_Trated" (
           $1                       := L 0.0,
           $2                       := "LightOnPump2");
      NOP   0;
NETWORK
TITLE =
      A     "Aux_LampPump2Fault";
      =     L 0.0;
      BLD   103;
      CALL  "Output_Trated" (
           $1                       := L 0.0,
           $2                       := "LightFaultPump2");
      NOP   0;
NETWORK
TITLE =
      A     "Aux_LampFan1On";
      =     L 0.0;
      BLD   103;
      CALL  "Output_Trated" (
           $1                       := L 0.0,
           $2                       := "LightOnFan1");
      NOP   0;
NETWORK
TITLE =
      A     "Aux_LampFan1Fault";
      =     L 0.0;
      BLD   103;
      CALL  "Output_Trated" (
           $1                       := L 0.0,
           $2                       := "LightFaultFan1");
      NOP   0;
NETWORK
TITLE =
      A     "Aux_LampFan2On";
      =     L 0.0;
      BLD   103;
      CALL  "Output_Trated" (
           $1                       := L 0.0,
           $2                       := "LightOnFan2");
      NOP   0;
NETWORK
TITLE =
      A     "Aux_LampFan2Fault";
      =     L 0.0;
      BLD   103;
      CALL  "Output_Trated" (
           $1                       := L 0.0,
           $2                       := "LightFaultFan2");
      NOP   0;
NETWORK
TITLE =
      A     "Aux_LampAdiabaticOn";
      =     L 0.0;
      BLD   103;
      CALL  "Output_Trated" (
           $1                       := L 0.0,
           $2                       := "LightOnAdb");
      NOP   0;
NETWORK
TITLE =
      A     "Aux_LampAdiabaticFault";
      =     L 0.0;
      BLD   103;
      CALL  "Output_Trated" (
           $1                       := L 0.0,
           $2                       := "LightFaultAdb");
      NOP   0;
END_FUNCTION

// FC 105: know-how protected block, not included

// FC 205: know-how protected block, not included

DATA_BLOCK "DBData"	// DB 1
VERSION : 0.1
  STRUCT
   setTempFan1 : REAL  := 3.500000e+001;
   setTempFan2 : REAL  := 3.700000e+001;
   setTempAdiabatic : REAL  := 4.200000e+001;
   histeresFan1 : REAL  := 2.000000e+000;
   histeresFan2 : REAL  := 2.000000e+000;
   histeresAdiabatic : REAL  := 2.000000e+000;
   setPump1On : BOOL  := TRUE;
   setPump2On : BOOL ;
   setPump12On : BOOL ;
   STAT9 : REAL ;
   alarmeReset : BOOL ;
   pump1Animated : BOOL ;
   pump2Animated : BOOL ;
   fan1Animated : BOOL ;
   fan2Animated : BOOL ;
   adiabaticAnimated : BOOL ;
   STAT16 : REAL ;
   STAT17 : REAL ;
   STAT18 : REAL ;
  END_STRUCT ;	
BEGIN
   setTempFan1 := 3.600000e+01;
   setTempFan2 := 3.900000e+01;
   setTempAdiabatic := 4.200000e+01;
   histeresFan1 := 2.000000e+00;
   histeresFan2 := 2.000000e+00;
   histeresAdiabatic := 2.000000e+00;
   setPump1On := TRUE;
   STAT9 := 4.700000e+01;
   alarmeReset := TRUE;
   pump1Animated := TRUE;
   fan1Animated := TRUE;
   STAT16 := 3.400000e+01;
   STAT17 := 3.700000e+01;
   STAT18 := 4.000000e+01;
END_DATA_BLOCK

DATA_BLOCK "DB_Alarm"	// DB 2
VERSION : 0.1
  STRUCT
   alarmSeries1 : WORD ;
   alarmSereis2 : WORD ;
  END_STRUCT ;	
BEGIN
   alarmSeries1 := W#16#90;
   alarmSereis2 := W#16#100;
END_DATA_BLOCK

DATA_BLOCK "Run Time Animation"	// DB 3
VERSION : 0.1
  STRUCT
   pump1OnAnimation : BOOL ;
   pump2OnAnimation : BOOL ;
   fan1OnAnimation : BOOL ;
   fan2OnAnimation : BOOL ;
   adiabaticOnAnimation : BOOL ;
   portugueseLanguage : BOOL  := TRUE;
   englishLanguage : BOOL ;
   bipolarScaling : BOOL ;
  END_STRUCT ;	
BEGIN
END_DATA_BLOCK

DATA_BLOCK "DBAnalog"	// DB 64
VERSION : 0.1
  STRUCT
   sensorAnalog1 : REAL ;
   sensorAnalog2 : REAL ;
   sensorAnalog3 : REAL ;
   sensorAnalog4 : REAL ;
   sensorAnalog5 : REAL ;
   sensorAnalog6 : REAL ;
   sensorAnalog7 : REAL ;
   sensorFactor1 : REAL  := 2.500000e+002;
   sensorFactor2 : REAL  := 2.500000e+002;
   sensorFactor3 : REAL  := 2.500000e+002;
   sensorFactor4 : REAL  := 2.500000e+002;
   sensorFactor5 : REAL  := 2.500000e+002;
   sensorFactor6 : REAL  := 2.500000e+002;
   sensorFactor7 : REAL  := 2.500000e+002;
  END_STRUCT ;	
BEGIN
   sensorAnalog1 := 3.506667e+01;
   sensorAnalog2 := 3.062500e+01;
   sensorFactor1 := 3.000000e+02;
   sensorFactor2 := 3.200000e+02;
END_DATA_BLOCK

ORGANIZATION_BLOCK "Cycle Execution"	// OB 1
VERSION : 0.1
VAR_TEMP
  TEMP0 : BYTE ;
  TEMP1 : BYTE ;
  TEMP2 : BYTE ;
  TEMP3 : BYTE ;
  TEMP4 : BYTE ;
  TEMP5 : BYTE ;
  TEMP6 : INT ;
  TEMP7 : INT ;
  TEMP8 : INT ;
  TEMP9 : DATE_AND_TIME ;
END_VAR
BEGIN
NETWORK
TITLE =
      CALL  "Tratamento_Inputs";
      NOP   0;
NETWORK
TITLE =
      CALL  "Tratamento Saida";
      NOP   0;
NETWORK
TITLE =
      CALL  "Pump_Logic";
      NOP   0;
NETWORK
TITLE =
      CALL  "Acionaqamento Ventilador";
      NOP   0;
NETWORK
TITLE =
      CALL  "Analog_Trated";
      NOP   0;
NETWORK
TITLE =
      CALL  FC 9;
      NOP   0;
NETWORK
TITLE =
      CALL  FC 95;
NETWORK
TITLE =
      CALL  "New Analog";
END_ORGANIZATION_BLOCK
